FUNCTION AddNums : INT
VAR_INPUT
	pNum : POINTER TO INT;
END_VAR
VAR
	ppNum : POINTER TO POINTER TO INT;
END_VAR


ppNum := ADR(pNum);
ppNum^^ := 25;

END_FUNCTION

(* stored: Version 1.1.0.1, ProductVersion 3.1.4024.16
   POU AddNums: Id {a995b3d7-7f8e-4745-80a7-aec1ee53f71a}, SpecialFunc None *)
